INTERFACE I_EM_DockingInterface

METHOD PUBLIC m_CloseDockingClamps : BOOL
END_METHOD

METHOD PUBLIC m_DockBox : BOOL
END_METHOD

METHOD PUBLIC m_OpenDockingClamps : BOOL
END_METHOD

METHOD PUBLIC m_UndockBox : BOOL
END_METHOD

PROPERTY PUBLIC p_bStaBoxAtDockedPosition : BOOL
GET
END_GET
END_PROPERTY

PROPERTY PUBLIC p_bStaBoxAtPreDockingPosition : BOOL
GET
END_GET
END_PROPERTY

PROPERTY p_bStaDockingClampsClosed : BOOL
GET
END_GET
END_PROPERTY

PROPERTY PUBLIC p_bStaDockingClampsOpened : BOOL
GET
END_GET
END_PROPERTY

PROPERTY PUBLIC p_bStaDockingDone : BOOL
GET
END_GET
END_PROPERTY

PROPERTY PUBLIC p_bStaDockingPositionFree : BOOL
GET
END_GET
END_PROPERTY

PROPERTY p_bStaUndockingDone : BOOL
GET
END_GET
END_PROPERTY

END_INTERFACE

(* stored: Version 1.1.0.1, ProductVersion 3.1.4024.12
   Itf I_EM_DockingInterface: Id {3ea93f09-d1a0-4ebe-babd-9e36271191c3}
   Method m_CloseDockingClamps: Id {a063fa03-5bc9-4219-92ac-a04138bab614}
   Method m_DockBox: Id {dca22798-0aaf-4b3c-846d-6df35f37a55a}
   Method m_OpenDockingClamps: Id {e676b370-a568-44cf-9f99-607fd70fa66e}
   Method m_UndockBox: Id {262ccc0e-85ee-4237-a109-3c6cef9168b3}
   Property p_bStaBoxAtDockedPosition: Id {d4202ebb-b511-4f6f-a657-c7c6ce5b2872}
   Get Get: Id {3e12d0f4-ac36-48f0-b54f-3258441d6784}
   Property p_bStaBoxAtPreDockingPosition: Id {981f9549-0fc6-4369-b4e5-6fd9571cb271}
   Get Get: Id {a60d4109-117a-4fd9-8906-294aa109f439}
   Property p_bStaDockingClampsClosed: Id {6d1ea4a4-bbc3-402d-8c34-066ff838f2b4}
   Get Get: Id {8836389a-1167-458d-9c81-577b2eab952f}
   Property p_bStaDockingClampsOpened: Id {954ef9eb-2f78-4314-9437-b5415faf2cf7}
   Get Get: Id {6ced54bd-7135-47b9-8981-7e1587500a2b}
   Property p_bStaDockingDone: Id {119a5edb-ffdb-4f4f-9343-3e394400ede1}
   Get Get: Id {17cc67f7-6672-4075-ac5a-c85b499c8d31}
   Property p_bStaDockingPositionFree: Id {c424f01b-55ae-42f0-8101-0a31e23b1a1c}
   Get Get: Id {e6ad4264-70df-4472-9506-a76001fa33be}
   Property p_bStaUndockingDone: Id {02715f9b-f1d8-4de7-9a05-f210f00a4cf0}
   Get Get: Id {5d7c2456-c1e4-49e6-97e0-da86fdd1a99a} *)
